(* LS Electric XG5000 project: 241008_연습문제3 *)
(* PLC LSPLC *)
(* module base 0 slot 0: 입력 모듈:XGI-D21A (DC 24V 입력, 8점 (전류소스/싱크입력)) *)
(* module base 0 slot 1: 출력 모듈:XGQ-RY1A (릴레이 출력, 8점 (2A용, 단독 COM.)) *)

PROGRAM NewProgram (* task: 스캔 프로그램 *)
VAR
    P1 AT %IX0.0.0 : BOOL;
    P10 AT %QX0.1.0 : BOOL;
    P2 AT %IX0.0.1 : BOOL;
    내부메모리 AT %MX0 : BOOL;
END_VAR

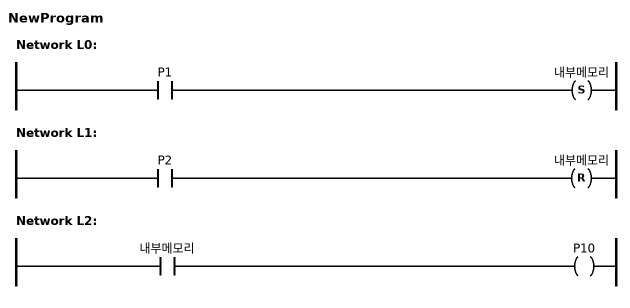
(* Rung L0 *)
IF P1 THEN 내부메모리 := TRUE; END_IF;
(* Rung L1 *)
IF P2 THEN 내부메모리 := FALSE; END_IF;
(* Rung L2 *)
P10 := 내부메모리;
END_PROGRAM